// SIMATIC STEP 7 (V5.x) project TEMA 13 EJERCICIO 28
// CPU: CPU313 C-2 DP(1)
// station: P_ADR_BUS
// station: Hardware
// station: Equipo SIMATIC 300
// program: Programa S7(1)

SYMBOL_TABLE
"FLANCOS"	DB 1	DB 1
"MANIOBRA"	DB 2	DB 2
"INTERMITENCIA"	FB 202	FB 202	// INTERMITENCIA CONFIGURABLE
"MARCHA"	I 0.0	BOOL
"PARO"	I 0.1	BOOL
"TERMICO"	I 0.2	BOOL
"Cycle Execution"	OB 1	OB 1
"MOTOR1"	Q 0.0	BOOL
"LEDMOTOR1"	Q 0.1	BOOL
"MOTOR2"	Q 0.2	BOOL
"LEDMOTOR2"	Q 0.3	BOOL
"LED PARO"	Q 0.4	BOOL
"LED AVERIA"	Q 0.5	BOOL
END_SYMBOL_TABLE

DATA_BLOCK "FLANCOS"	// DB 1
VERSION : 0.1
  STRUCT
   M0 : BOOL ;
   M1 : BOOL ;
   M2 : BOOL ;
   M3 : BOOL ;
   M4 : BOOL ;
   M5 : BOOL ;
   M6 : BOOL ;
   M7 : BOOL ;
   M10 : BOOL ;
   M11 : BOOL ;
   M12 : BOOL ;
   M13 : BOOL ;
   M14 : BOOL ;
   M15 : BOOL ;
   M16 : BOOL ;
   M17 : BOOL ;
   M20 : BOOL ;
   M21 : BOOL ;
   M22 : BOOL ;
   M23 : BOOL ;
   M24 : BOOL ;
   M25 : BOOL ;
   M26 : BOOL ;
   M27 : BOOL ;
  END_STRUCT ;	
BEGIN
END_DATA_BLOCK

DATA_BLOCK "MANIOBRA"	// DB 2
VERSION : 0.1
  STRUCT
   MARCA0 : BOOL ;
   MARCA1 : BOOL ;
   MARCA2 : BOOL ;
   MARCA3 : BOOL ;
   MARCA4 : BOOL ;
   MARCA5 : BOOL ;
   MARCA6 : BOOL ;
   MARCA7 : BOOL ;
   MARCA10 : BOOL ;
   MARCA11 : BOOL ;
   MARCA12 : BOOL ;
   MARCA13 : BOOL ;
   MARCA14 : BOOL ;
   MARCA15 : BOOL ;
   MARCA16 : BOOL ;
   MARCA17 : BOOL ;
  END_STRUCT ;	
BEGIN
END_DATA_BLOCK

ORGANIZATION_BLOCK "Cycle Execution"	// OB 1
TITLE = "Main Program Sweep (Cycle)"
//ARRANQUE INTERMITENTE DE 2 MOTORES
VERSION : 0.1
VAR_TEMP
  OB1_EV_CLASS : BYTE ;	//Bits 0-3 = 1 (Coming event), Bits 4-7 = 1 (Event class 1)
  OB1_SCAN_1 : BYTE ;	//1 (Cold restart scan 1 of OB 1), 3 (Scan 2-n of OB 1)
  OB1_PRIORITY : BYTE ;	//Priority of OB Execution
  OB1_OB_NUMBR : BYTE ;	//1 (Organization block 1, OB1)
  OB1_RESERVED_1 : BYTE ;	//Reserved for system
  OB1_RESERVED_2 : BYTE ;	//Reserved for system
  OB1_PREV_CYCLE : INT ;	//Cycle time of previous OB1 scan (milliseconds)
  OB1_MIN_CYCLE : INT ;	//Minimum cycle time of OB1 (milliseconds)
  OB1_MAX_CYCLE : INT ;	//Maximum cycle time of OB1 (milliseconds)
  OB1_DATE_TIME : DATE_AND_TIME ;	//Date and time OB1 started
END_VAR
BEGIN
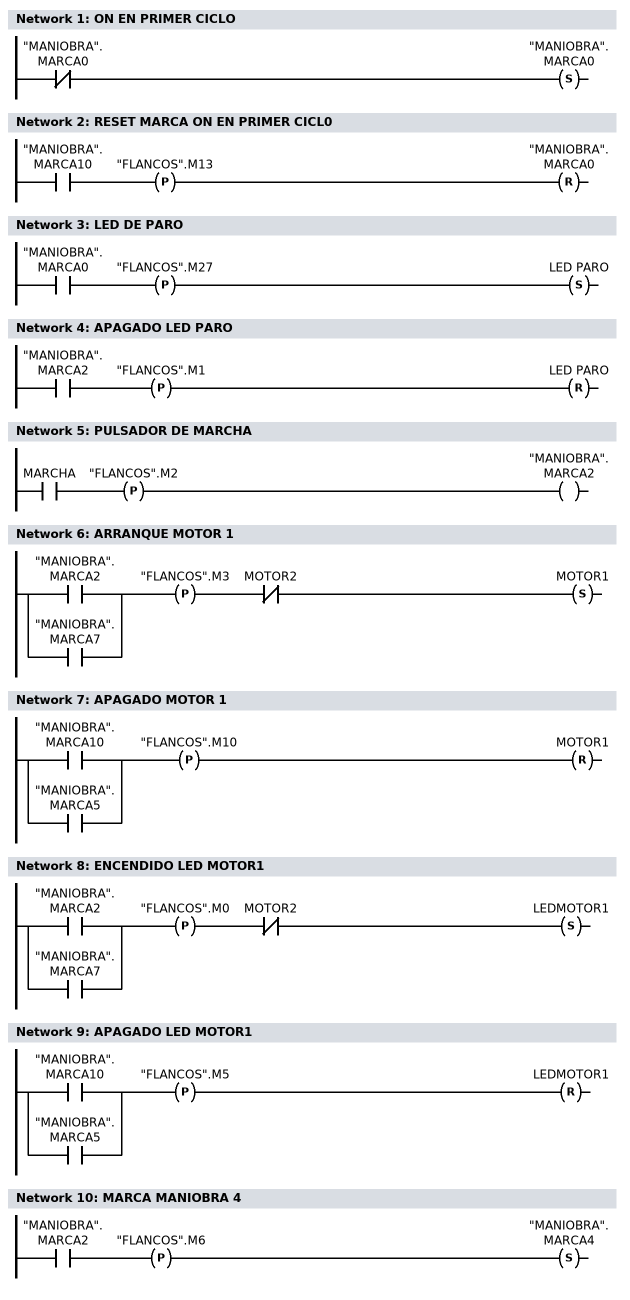
NETWORK
TITLE = ON EN PRIMER CICLO
      AN    "MANIOBRA".MARCA0;
      S     "MANIOBRA".MARCA0;
NETWORK
TITLE = RESET MARCA ON EN PRIMER CICL0
      A     "MANIOBRA".MARCA10;
      FP    "FLANCOS".M13;
      R     "MANIOBRA".MARCA0;
NETWORK
TITLE = LED DE PARO
      A     "MANIOBRA".MARCA0;
      FP    "FLANCOS".M27;
      S     "LED PARO";
NETWORK
TITLE = APAGADO LED PARO
      A     "MANIOBRA".MARCA2;
      FP    "FLANCOS".M1;
      R     "LED PARO";
NETWORK
TITLE = PULSADOR DE MARCHA
      A     "MARCHA";
      FP    "FLANCOS".M2;
      =     "MANIOBRA".MARCA2;
NETWORK
TITLE = ARRANQUE MOTOR 1 
      A(;
      O     "MANIOBRA".MARCA2;
      O     "MANIOBRA".MARCA7;
      );
      FP    "FLANCOS".M3;
      AN    "MOTOR2";
      S     "MOTOR1";
NETWORK
TITLE = APAGADO MOTOR 1 
//CONTACTO TEMPORIZADO TO APAGA MOTOR 1 
      A(;
      O     "MANIOBRA".MARCA10;
      O     "MANIOBRA".MARCA5;
      );
      FP    "FLANCOS".M10;
      R     "MOTOR1";
NETWORK
TITLE = ENCENDIDO LED MOTOR1
      A(;
      O     "MANIOBRA".MARCA2;
      O     "MANIOBRA".MARCA7;
      );
      FP    "FLANCOS".M0;
      AN    "MOTOR2";
      S     "LEDMOTOR1";
NETWORK
TITLE = APAGADO LED MOTOR1
      A(;
      O     "MANIOBRA".MARCA10;
      O     "MANIOBRA".MARCA5;
      );
      FP    "FLANCOS".M5;
      R     "LEDMOTOR1";
NETWORK
TITLE = MARCA MANIOBRA 4
//ESTA MARCA NOS MANTENDRA EL FLUJO DE CORRIENTE ININTERRUMPIDA PARA LA 
//ALIMENTACION DE LOS TEMPORIZADORES DE INTERMITENCIA.
      A     "MANIOBRA".MARCA2;
      FP    "FLANCOS".M6;
      S     "MANIOBRA".MARCA4;
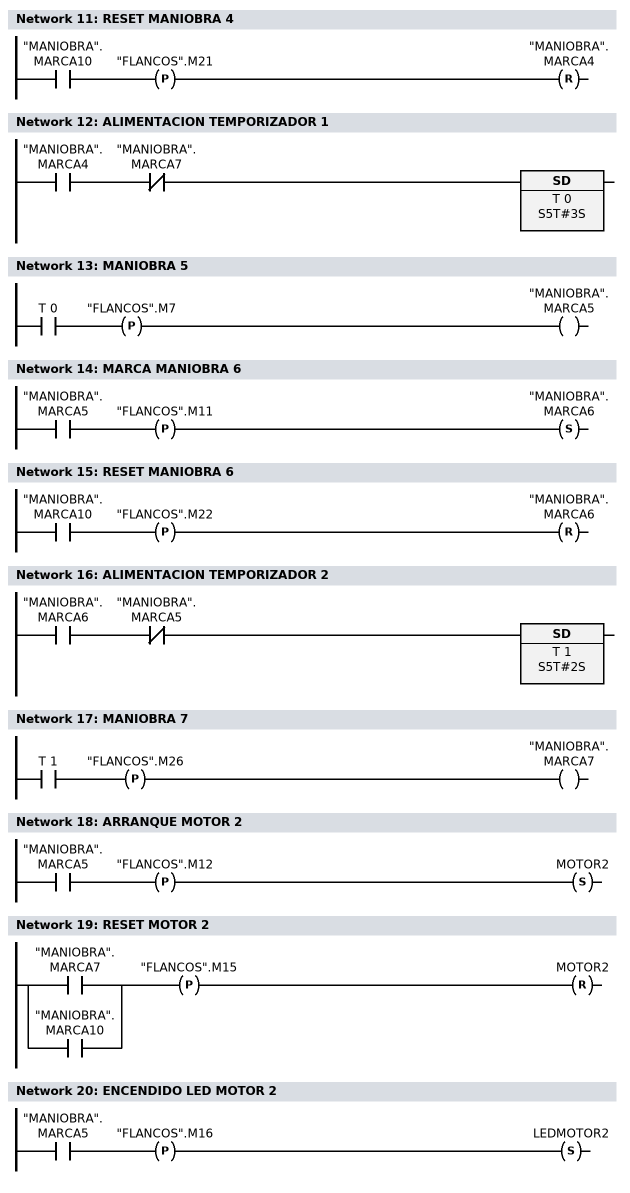
NETWORK
TITLE = RESET MANIOBRA 4 
      A     "MANIOBRA".MARCA10;
      FP    "FLANCOS".M21;
      R     "MANIOBRA".MARCA4;
NETWORK
TITLE = ALIMENTACION TEMPORIZADOR 1 
      A     "MANIOBRA".MARCA4;
      AN    "MANIOBRA".MARCA7;
      L     S5T#3S;
      SD    T 0;
NETWORK
TITLE = MANIOBRA 5 
      A     T 0;
      FP    "FLANCOS".M7;
      =     "MANIOBRA".MARCA5;
NETWORK
TITLE = MARCA MANIOBRA 6
//DESARROLLA LA MISMA FUNCION QUE LA MENCIONADA ANTERIORMENTE
      A     "MANIOBRA".MARCA5;
      FP    "FLANCOS".M11;
      S     "MANIOBRA".MARCA6;
NETWORK
TITLE = RESET MANIOBRA 6
      A     "MANIOBRA".MARCA10;
      FP    "FLANCOS".M22;
      R     "MANIOBRA".MARCA6;
NETWORK
TITLE = ALIMENTACION TEMPORIZADOR 2 
      A     "MANIOBRA".MARCA6;
      AN    "MANIOBRA".MARCA5;
      L     S5T#2S;
      SD    T 1;
NETWORK
TITLE = MANIOBRA 7
      A     T 1;
      FP    "FLANCOS".M26;
      =     "MANIOBRA".MARCA7;
NETWORK
TITLE = ARRANQUE MOTOR 2 
      A     "MANIOBRA".MARCA5;
      FP    "FLANCOS".M12;
      S     "MOTOR2";
NETWORK
TITLE = RESET MOTOR 2
      A(;
      O     "MANIOBRA".MARCA7;
      O     "MANIOBRA".MARCA10;
      );
      FP    "FLANCOS".M15;
      R     "MOTOR2";
NETWORK
TITLE = ENCENDIDO LED MOTOR 2 
      A     "MANIOBRA".MARCA5;
      FP    "FLANCOS".M16;
      S     "LEDMOTOR2";
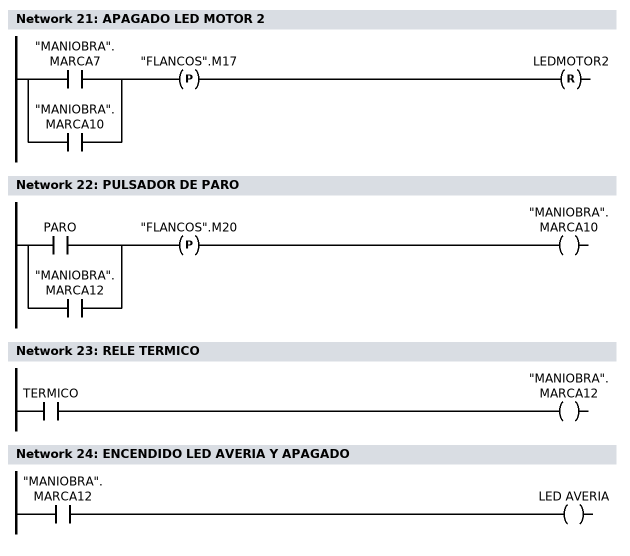
NETWORK
TITLE = APAGADO LED MOTOR 2 
      A(;
      O     "MANIOBRA".MARCA7;
      O     "MANIOBRA".MARCA10;
      );
      FP    "FLANCOS".M17;
      R     "LEDMOTOR2";
NETWORK
TITLE = PULSADOR DE PARO
      A(;
      O     "PARO";
      O     "MANIOBRA".MARCA12;
      );
      FP    "FLANCOS".M20;
      =     "MANIOBRA".MARCA10;
NETWORK
TITLE = RELE TERMICO
      A     "TERMICO";
      =     "MANIOBRA".MARCA12;
NETWORK
TITLE = ENCENDIDO LED AVERIA Y APAGADO
//COMO ES UNA SIMULACION EL TIEMPO QUE ESTE EL PULSADOR EN ON LO ESTARA EL LED
      A     "MANIOBRA".MARCA12;
      =     "LED AVERIA";
END_ORGANIZATION_BLOCK
